// TIA Portal V15.1 export
// export: Created 2020-06-12T07:35:40.5849609Z, ExportSetting None, DisplayName Totally Integrated Automation Portal, DisplayVersion V15.1, DisplayName TIA Portal Openness, DisplayVersion V15.1, DisplayName STEP 7 Professional, DisplayVersion V15.1, DisplayName STEP 7 Safety, DisplayVersion V15.1, DisplayName WinCC Advanced, DisplayVersion V15.1
FUNCTION_BLOCK "F_call"   // FB3, F_FBD
TITLE = Failsafe MAIN program
{ S7_Optimized_Access := 'TRUE' }
   VAR
      emst_del_reset { ExternalAccessible := 'False'; ExternalVisible := 'False'; ExternalWritable := 'False'} : Bool;   // EmStop delayed reset
      ESTOP { ExternalAccessible := 'False'; ExternalVisible := 'False'; ExternalWritable := 'False'} : ESTOP1;
      ACK { ExternalAccessible := 'False'; ExternalVisible := 'False'; ExternalWritable := 'False'} : ACK_GL;
      SD1_TOF { ExternalAccessible := 'False'; ExternalVisible := 'False'; ExternalWritable := 'False'} : TOF;
      RS_TON { ExternalAccessible := 'False'; ExternalVisible := 'False'; ExternalWritable := 'False'} : TON;
      FBACK_EMER_UNDEL { ExternalAccessible := 'False'; ExternalVisible := 'False'; ExternalWritable := 'False'} : FDBACK;
      FBACK_EMER_DEL { ExternalAccessible := 'False'; ExternalVisible := 'False'; ExternalWritable := 'False'} : FDBACK;
      FBACK_ES1LE1_EV02 { ExternalAccessible := 'False'; ExternalVisible := 'False'; ExternalWritable := 'False'} : FDBACK;
      FBACK_ES1LE1_M01 { ExternalAccessible := 'False'; ExternalVisible := 'False'; ExternalWritable := 'False'} : FDBACK;
      FBACK_ES1LE1_M01STO { ExternalAccessible := 'False'; ExternalVisible := 'False'; ExternalWritable := 'False'} : FDBACK;
      FBACK_ES1LE2_M01 { ExternalAccessible := 'False'; ExternalVisible := 'False'; ExternalWritable := 'False'} : FDBACK;
      FBACK_ES1LE2_M02 { ExternalAccessible := 'False'; ExternalVisible := 'False'; ExternalWritable := 'False'} : FDBACK;
      FBACK_ES1LE3_M01 { ExternalAccessible := 'False'; ExternalVisible := 'False'; ExternalWritable := 'False'} : FDBACK;
      FBACK_ES1LE3_M01STO { ExternalAccessible := 'False'; ExternalVisible := 'False'; ExternalWritable := 'False'} : FDBACK;
      FBACK_ES1LE4_EV01 { ExternalAccessible := 'False'; ExternalVisible := 'False'; ExternalWritable := 'False'} : FDBACK;
      FBACK_ES1LE4_EV02 { ExternalAccessible := 'False'; ExternalVisible := 'False'; ExternalWritable := 'False'} : FDBACK;
      FBACK_ES1LE4_M01 { ExternalAccessible := 'False'; ExternalVisible := 'False'; ExternalWritable := 'False'} : FDBACK;
      FBACK_ES1LE4_M01STO { ExternalAccessible := 'False'; ExternalVisible := 'False'; ExternalWritable := 'False'} : FDBACK;
      FBACK_ES1LM1_EV01 { ExternalAccessible := 'False'; ExternalVisible := 'False'; ExternalWritable := 'False'} : FDBACK;
      FBACK_ES1LM2_EV01 { ExternalAccessible := 'False'; ExternalVisible := 'False'; ExternalWritable := 'False'} : FDBACK;
      FBACK_ES1LS1_XS01 { ExternalAccessible := 'False'; ExternalVisible := 'False'; ExternalWritable := 'False'} : FDBACK;
      TOF_GYxx { ExternalAccessible := 'False'; ExternalVisible := 'False'; ExternalWritable := 'False'} : TOF;
      TOF_hood { ExternalAccessible := 'False'; ExternalVisible := 'False'; ExternalWritable := 'False'} : TOF;
      TOF_mcb { ExternalAccessible := 'False'; ExternalVisible := 'False'; ExternalWritable := 'False'} : TOF;
      TOF_trafo { ExternalAccessible := 'False'; ExternalVisible := 'False'; ExternalWritable := 'False'} : TOF;
      TMR_S43_flt { ExternalAccessible := 'False'; ExternalVisible := 'False'; ExternalWritable := 'False'} : TON;
      TMR_S43_auto { ExternalAccessible := 'False'; ExternalVisible := 'False'; ExternalWritable := 'False'} : TOF;
   END_VAR
   VAR_TEMP
      _area_safe : Bool;
      _hood_is_closed : Bool;
      _reset : Bool;
      _del_reset : Bool;
      _GD01_S43_flt : Bool;
      _GD01_S43_off : Bool;
      _GD01_S43_auto : Bool;
   END_VAR
BEGIN

REGION Network 1: Delayed automatic reset by GD01-S34 (timeout)
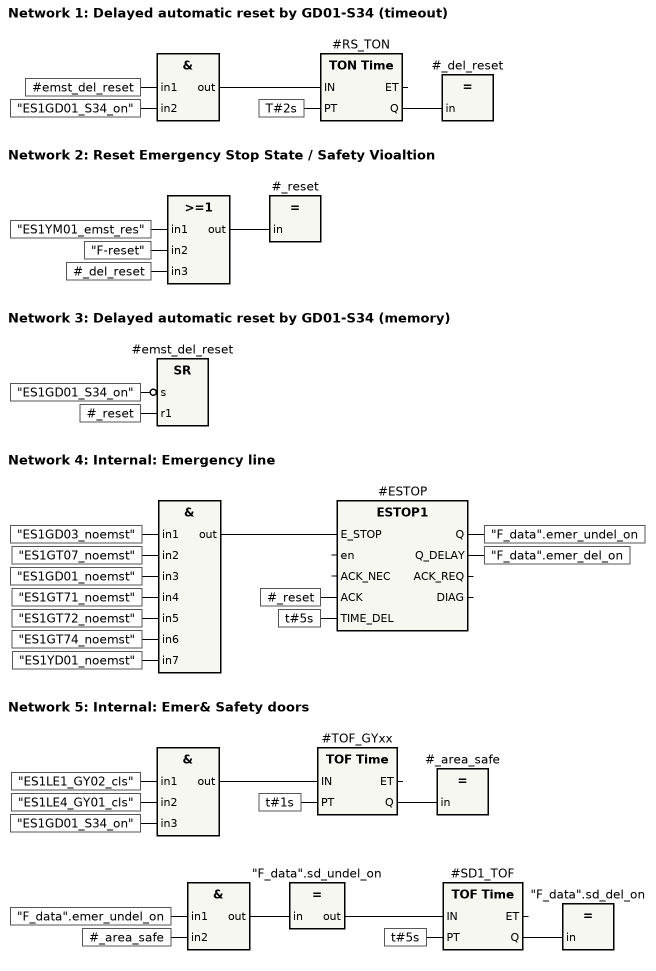
   #RS_TON.TON(IN := #emst_del_reset AND "ES1GD01_S34_on", PT := T#2s);
   #_del_reset := #RS_TON.Q;
END_REGION

REGION Network 2: Reset Emergency Stop State / Safety Vioaltion
   #_reset := "ES1YM01_emst_res" OR "F-reset" OR #_del_reset;
END_REGION

REGION Network 3: Delayed automatic reset by GD01-S34 (memory)
   IF NOT "ES1GD01_S34_on" THEN
       #emst_del_reset := TRUE;   // SR flip-flop
   END_IF;
   IF #_reset THEN #emst_del_reset := FALSE; END_IF;
END_REGION

REGION Network 4: Internal: Emergency line
   #ESTOP(E_STOP := "ES1GD03_noemst" AND "ES1GT07_noemst" AND "ES1GD01_noemst" AND "ES1GT71_noemst" AND "ES1GT72_noemst" AND "ES1GT74_noemst" AND "ES1YD01_noemst",   // ESTOP1
          ACK := #_reset,
          TIME_DEL := t#5s,
          Q => "F_data".emer_undel_on,
          Q_DELAY => "F_data".emer_del_on);
END_REGION

REGION Network 5: Internal: Emer& Safety doors
   // ES1LE1.GY02 = top platfromr safety door
   // ES1LE4.GY01 = portal ladder
   #TOF_GYxx.TOF(IN := "ES1LE1_GY02_cls" AND "ES1LE4_GY01_cls" AND "ES1GD01_S34_on", PT := t#1s);
   #_area_safe := #TOF_GYxx.Q;
   "F_data".sd_undel_on := "F_data".emer_undel_on AND #_area_safe;
   #SD1_TOF.TOF(IN := "F_data".sd_undel_on, PT := t#5s);
   "F_data".sd_del_on := #SD1_TOF.Q;
END_REGION

REGION Network 6: ES1GD01-S43 treat
   // The switch S43 has non-ideal switching: the signal between positions are all 0
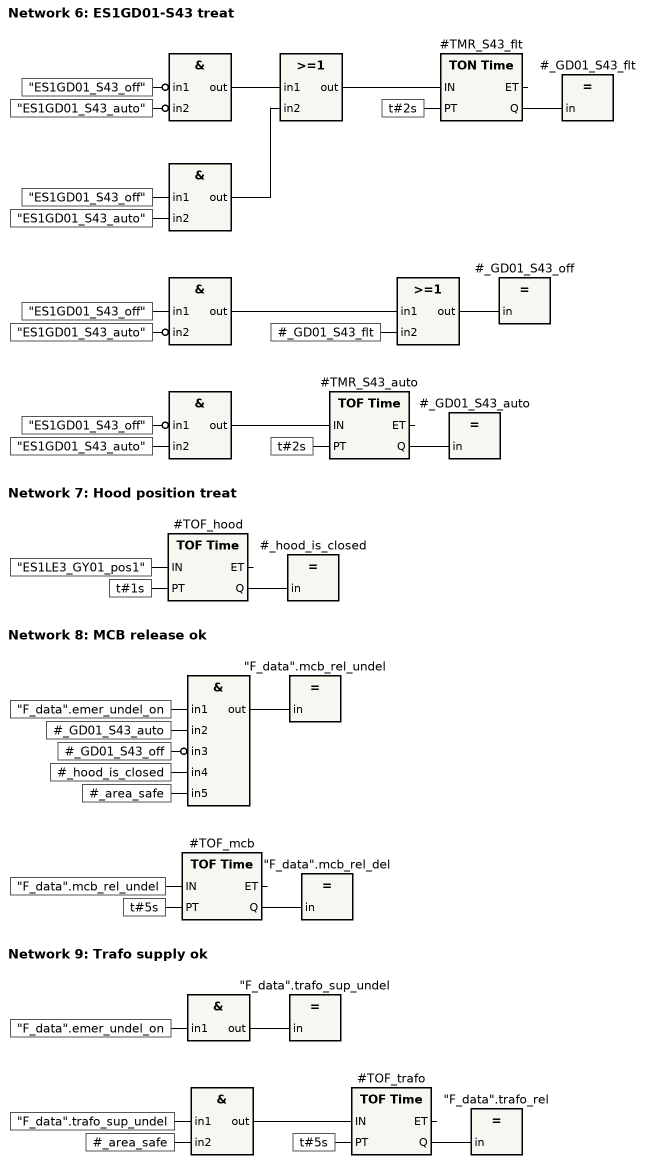
   #TMR_S43_flt.TON(IN := (NOT "ES1GD01_S43_off" AND NOT "ES1GD01_S43_auto") OR ("ES1GD01_S43_off" AND "ES1GD01_S43_auto"),
                    PT := t#2s);
   #_GD01_S43_flt := #TMR_S43_flt.Q;
   #_GD01_S43_off := ("ES1GD01_S43_off" AND NOT "ES1GD01_S43_auto") OR #_GD01_S43_flt;
   #TMR_S43_auto.TOF(IN := NOT "ES1GD01_S43_off" AND "ES1GD01_S43_auto", PT := t#2s);
   #_GD01_S43_auto := #TMR_S43_auto.Q;
END_REGION

REGION Network 7: Hood position treat
   #TOF_hood.TOF(IN := "ES1LE3_GY01_pos1", PT := t#1s);
   #_hood_is_closed := #TOF_hood.Q;
END_REGION

REGION Network 8: MCB release ok
   "F_data".mcb_rel_undel := "F_data".emer_undel_on AND #_GD01_S43_auto AND NOT #_GD01_S43_off AND #_hood_is_closed AND #_area_safe;
   #TOF_mcb.TOF(IN := "F_data".mcb_rel_undel, PT := t#5s);
   "F_data".mcb_rel_del := #TOF_mcb.Q;
END_REGION

REGION Network 9: Trafo supply ok
   "F_data".trafo_sup_undel := "F_data".emer_undel_on;
   #TOF_trafo.TOF(IN := "F_data".trafo_sup_undel AND #_area_safe, PT := t#5s);
   "F_data".trafo_rel := #TOF_trafo.Q;
END_REGION

REGION Network 10: Out: Emergency line Undelayed
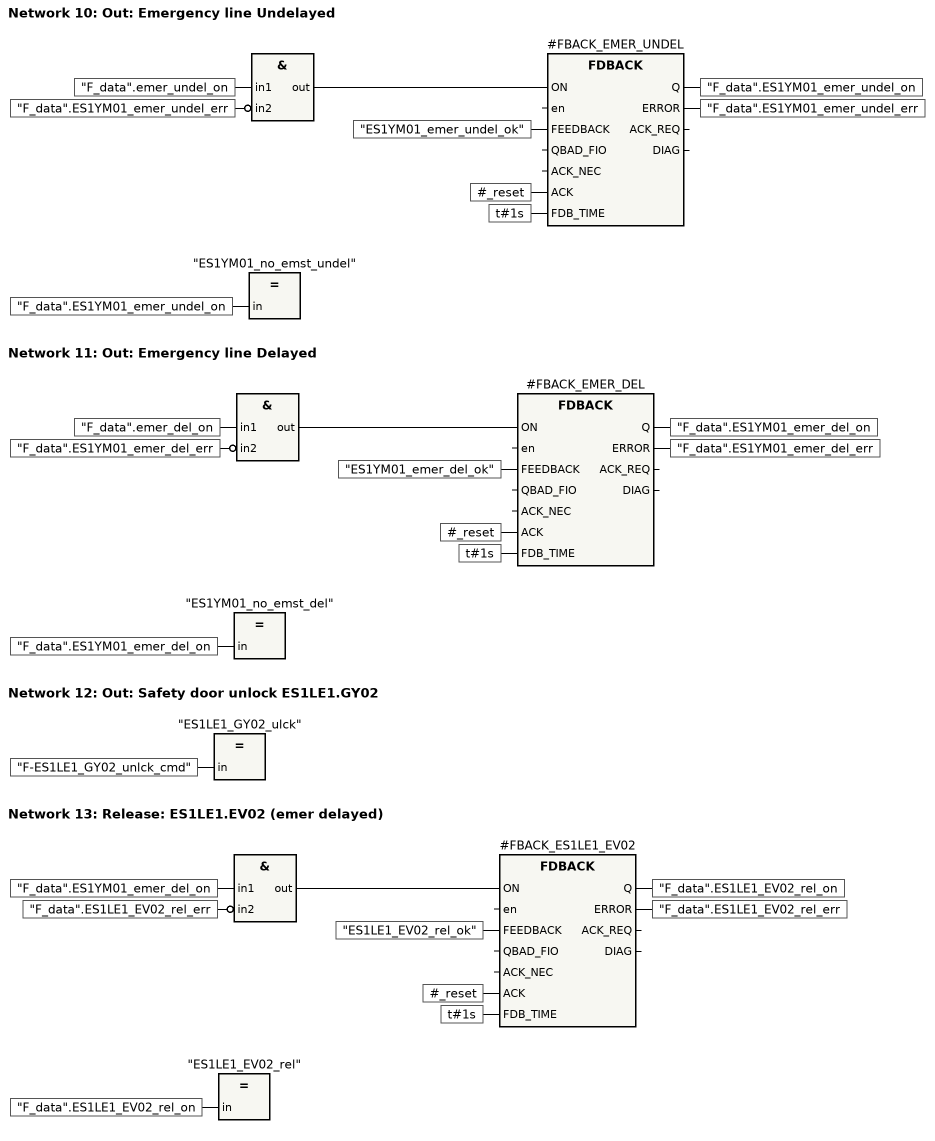
   #FBACK_EMER_UNDEL(ON := "F_data".emer_undel_on AND NOT "F_data".ES1YM01_emer_undel_err,   // FDBACK
                     FEEDBACK := "ES1YM01_emer_undel_ok",
                     ACK := #_reset,
                     FDB_TIME := t#1s,
                     Q => "F_data".ES1YM01_emer_undel_on,
                     ERROR => "F_data".ES1YM01_emer_undel_err);
   "ES1YM01_no_emst_undel" := "F_data".ES1YM01_emer_undel_on;
END_REGION

REGION Network 11: Out: Emergency line Delayed
   #FBACK_EMER_DEL(ON := "F_data".emer_del_on AND NOT "F_data".ES1YM01_emer_del_err,   // FDBACK
                   FEEDBACK := "ES1YM01_emer_del_ok",
                   ACK := #_reset,
                   FDB_TIME := t#1s,
                   Q => "F_data".ES1YM01_emer_del_on,
                   ERROR => "F_data".ES1YM01_emer_del_err);
   "ES1YM01_no_emst_del" := "F_data".ES1YM01_emer_del_on;
END_REGION

REGION Network 12: Out: Safety door unlock ES1LE1.GY02
   "ES1LE1_GY02_ulck" := "F-ES1LE1_GY02_unlck_cmd";
END_REGION

REGION Network 13: Release: ES1LE1.EV02 (emer delayed)
   #FBACK_ES1LE1_EV02(ON := "F_data".ES1YM01_emer_del_on AND NOT "F_data".ES1LE1_EV02_rel_err,   // FDBACK
                      FEEDBACK := "ES1LE1_EV02_rel_ok",
                      ACK := #_reset,
                      FDB_TIME := t#1s,
                      Q => "F_data".ES1LE1_EV02_rel_on,
                      ERROR => "F_data".ES1LE1_EV02_rel_err);
   "ES1LE1_EV02_rel" := "F_data".ES1LE1_EV02_rel_on;
END_REGION

REGION Network 14: Release: ES1LE4.EV01 (emer delayed)
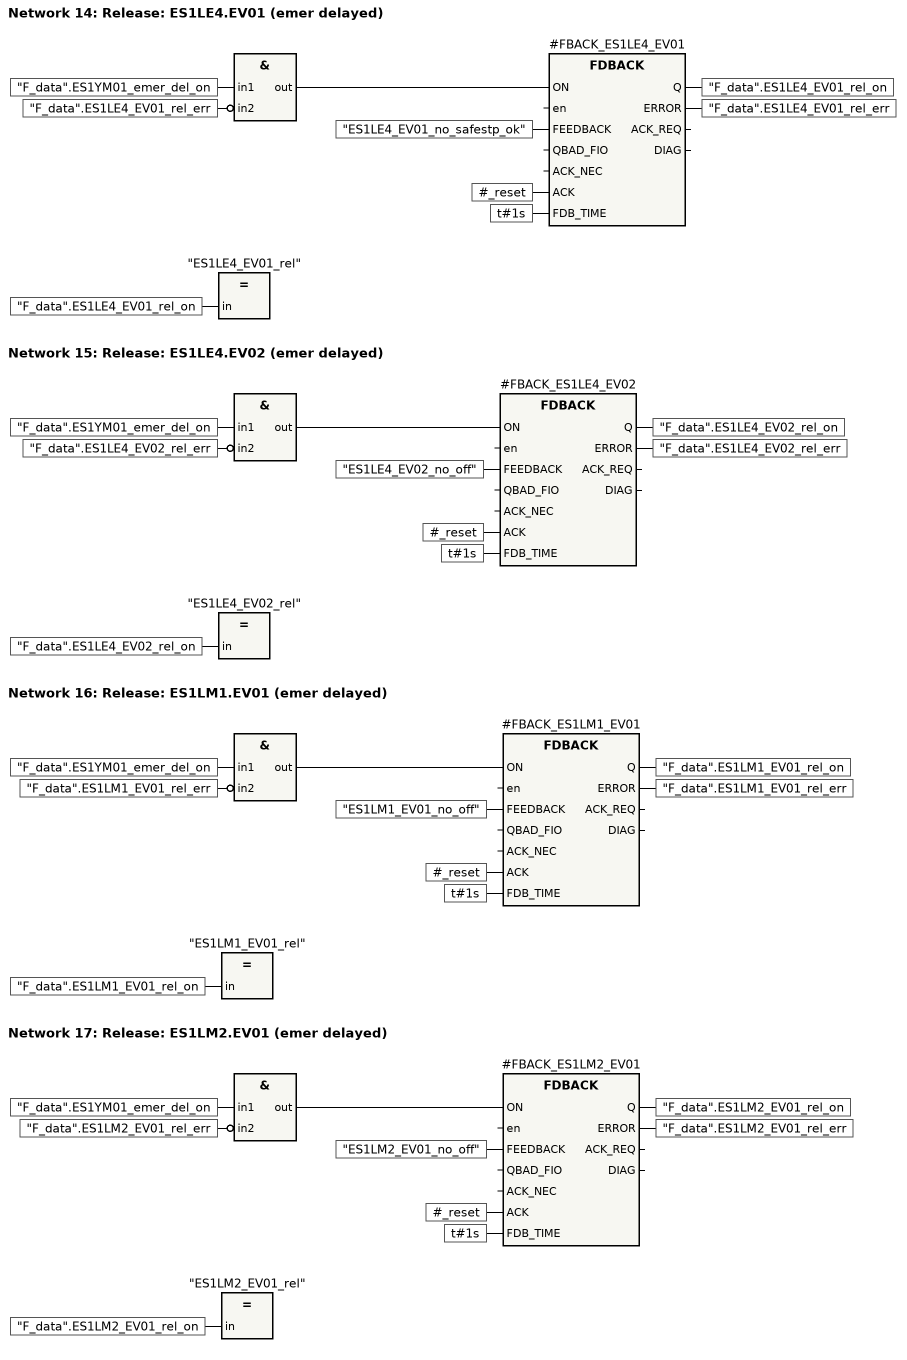
   #FBACK_ES1LE4_EV01(ON := "F_data".ES1YM01_emer_del_on AND NOT "F_data".ES1LE4_EV01_rel_err,   // FDBACK
                      FEEDBACK := "ES1LE4_EV01_no_safestp_ok",
                      ACK := #_reset,
                      FDB_TIME := t#1s,
                      Q => "F_data".ES1LE4_EV01_rel_on,
                      ERROR => "F_data".ES1LE4_EV01_rel_err);
   "ES1LE4_EV01_rel" := "F_data".ES1LE4_EV01_rel_on;
END_REGION

REGION Network 15: Release: ES1LE4.EV02 (emer delayed)
   #FBACK_ES1LE4_EV02(ON := "F_data".ES1YM01_emer_del_on AND NOT "F_data".ES1LE4_EV02_rel_err,   // FDBACK
                      FEEDBACK := "ES1LE4_EV02_no_off",
                      ACK := #_reset,
                      FDB_TIME := t#1s,
                      Q => "F_data".ES1LE4_EV02_rel_on,
                      ERROR => "F_data".ES1LE4_EV02_rel_err);
   "ES1LE4_EV02_rel" := "F_data".ES1LE4_EV02_rel_on;
END_REGION

REGION Network 16: Release: ES1LM1.EV01 (emer delayed)
   #FBACK_ES1LM1_EV01(ON := "F_data".ES1YM01_emer_del_on AND NOT "F_data".ES1LM1_EV01_rel_err,   // FDBACK
                      FEEDBACK := "ES1LM1_EV01_no_off",
                      ACK := #_reset,
                      FDB_TIME := t#1s,
                      Q => "F_data".ES1LM1_EV01_rel_on,
                      ERROR => "F_data".ES1LM1_EV01_rel_err);
   "ES1LM1_EV01_rel" := "F_data".ES1LM1_EV01_rel_on;
END_REGION

REGION Network 17: Release: ES1LM2.EV01 (emer delayed)
   #FBACK_ES1LM2_EV01(ON := "F_data".ES1YM01_emer_del_on AND NOT "F_data".ES1LM2_EV01_rel_err,   // FDBACK
                      FEEDBACK := "ES1LM2_EV01_no_off",
                      ACK := #_reset,
                      FDB_TIME := t#1s,
                      Q => "F_data".ES1LM2_EV01_rel_on,
                      ERROR => "F_data".ES1LM2_EV01_rel_err);
   "ES1LM2_EV01_rel" := "F_data".ES1LM2_EV01_rel_on;
END_REGION

REGION Network 18: Release: ES1LE1.M01 (emer undelayed)
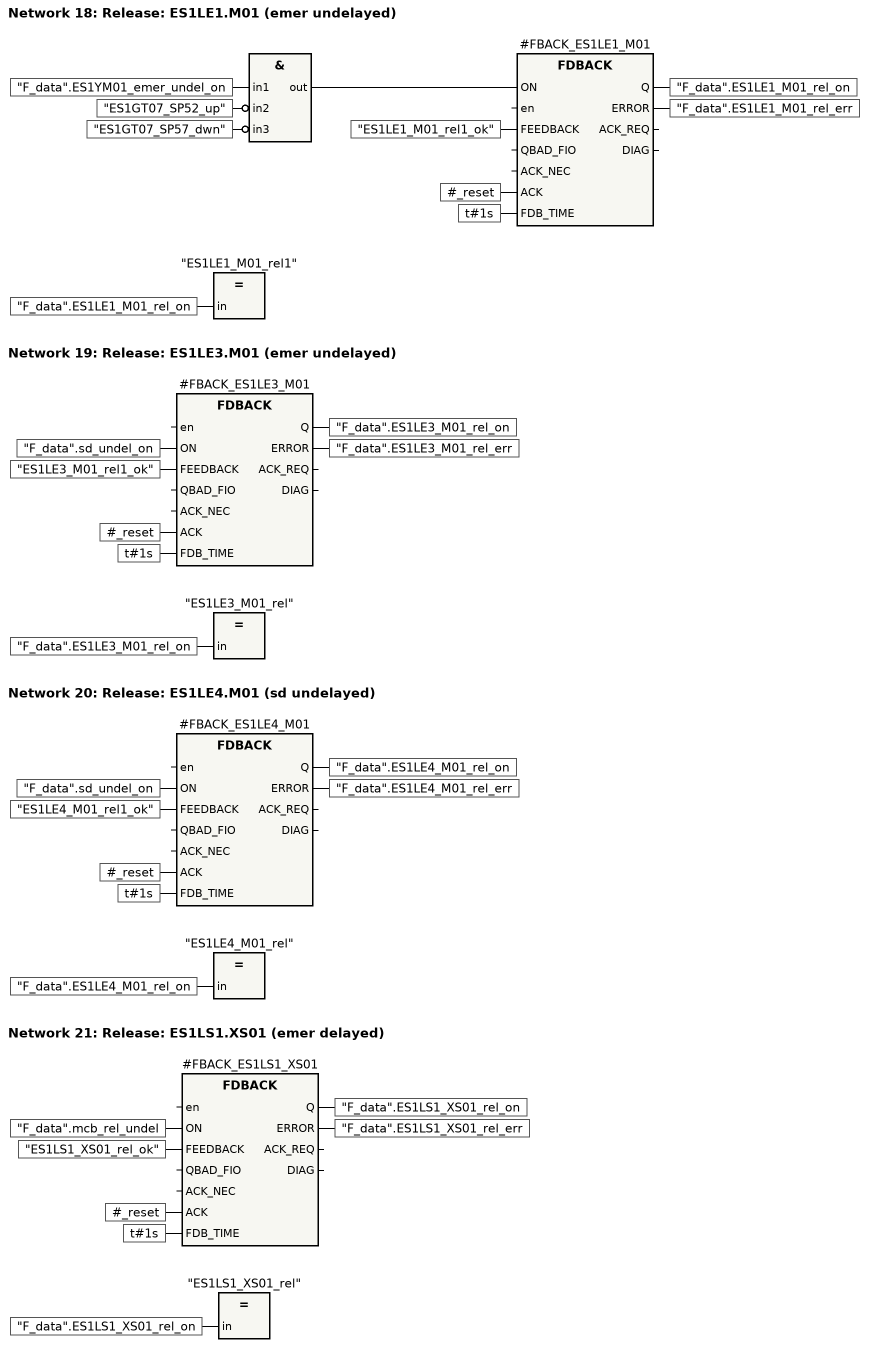
   #FBACK_ES1LE1_M01(ON := "F_data".ES1YM01_emer_undel_on AND NOT "ES1GT07_SP52_up" AND NOT "ES1GT07_SP57_dwn",   // FDBACK
                     FEEDBACK := "ES1LE1_M01_rel1_ok",
                     ACK := #_reset,
                     FDB_TIME := t#1s,
                     Q => "F_data".ES1LE1_M01_rel_on,
                     ERROR => "F_data".ES1LE1_M01_rel_err);
   "ES1LE1_M01_rel1" := "F_data".ES1LE1_M01_rel_on;
END_REGION

REGION Network 19: Release: ES1LE3.M01 (emer undelayed)
   #FBACK_ES1LE3_M01(ON := "F_data".sd_undel_on,   // FDBACK
                     FEEDBACK := "ES1LE3_M01_rel1_ok",
                     ACK := #_reset,
                     FDB_TIME := t#1s,
                     Q => "F_data".ES1LE3_M01_rel_on,
                     ERROR => "F_data".ES1LE3_M01_rel_err);
   "ES1LE3_M01_rel" := "F_data".ES1LE3_M01_rel_on;
END_REGION

REGION Network 20: Release: ES1LE4.M01 (sd undelayed)
   #FBACK_ES1LE4_M01(ON := "F_data".sd_undel_on,   // FDBACK
                     FEEDBACK := "ES1LE4_M01_rel1_ok",
                     ACK := #_reset,
                     FDB_TIME := t#1s,
                     Q => "F_data".ES1LE4_M01_rel_on,
                     ERROR => "F_data".ES1LE4_M01_rel_err);
   "ES1LE4_M01_rel" := "F_data".ES1LE4_M01_rel_on;
END_REGION

REGION Network 21: Release: ES1LS1.XS01 (emer delayed)
   #FBACK_ES1LS1_XS01(ON := "F_data".mcb_rel_undel,   // FDBACK
                      FEEDBACK := "ES1LS1_XS01_rel_ok",
                      ACK := #_reset,
                      FDB_TIME := t#1s,
                      Q => "F_data".ES1LS1_XS01_rel_on,
                      ERROR => "F_data".ES1LS1_XS01_rel_err);
   "ES1LS1_XS01_rel" := "F_data".ES1LS1_XS01_rel_on;
END_REGION

REGION Network 22: Release ES1LT1.XS01/no_emst (emer undelayed)
   // !! WARNING! 
   // PuM/2018-08-13: This E-STOP is not in SafetyMatrix and it has only one line (not two as required). Because of that I implement only local emeregecny stop.
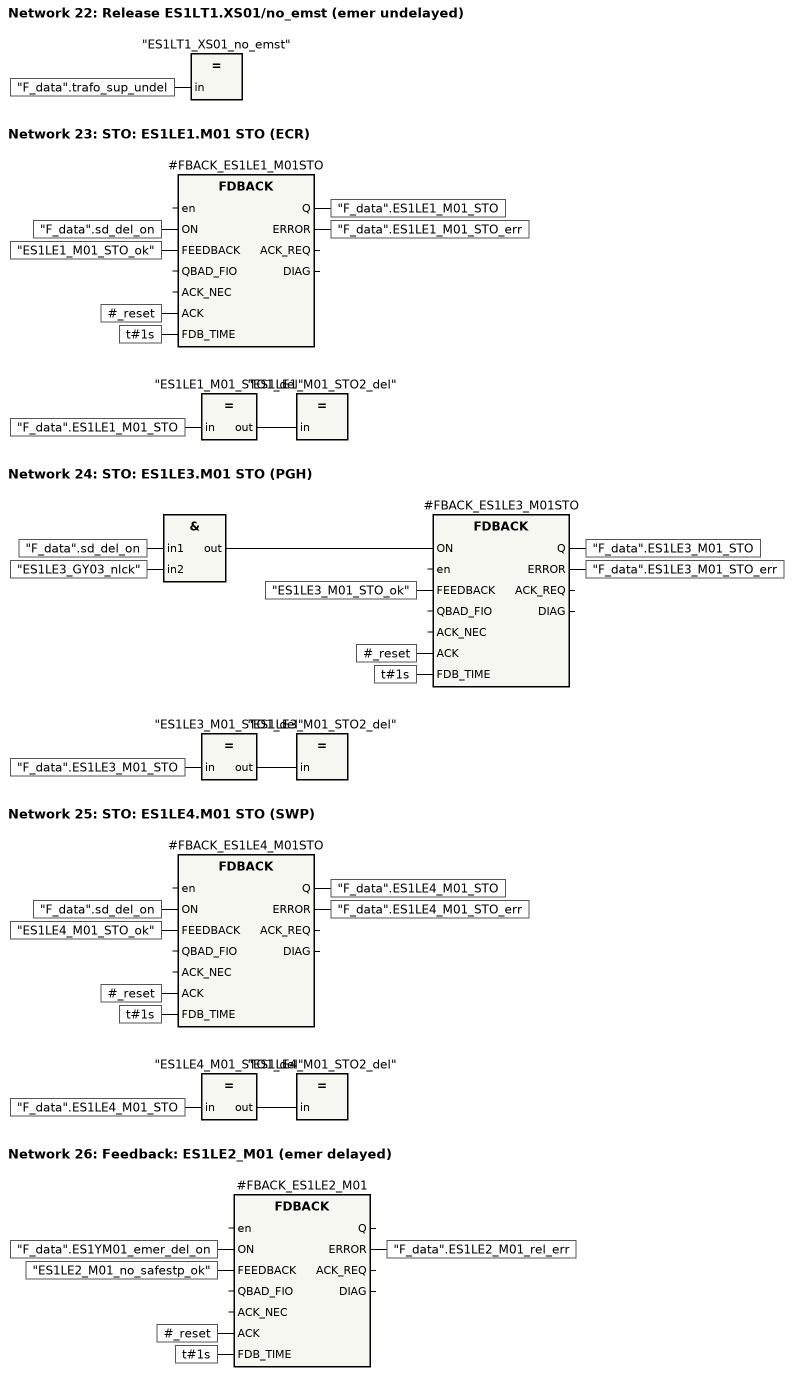
   "ES1LT1_XS01_no_emst" := "F_data".trafo_sup_undel;
END_REGION

REGION Network 23: STO: ES1LE1.M01 STO (ECR)
   #FBACK_ES1LE1_M01STO(ON := "F_data".sd_del_on,   // FDBACK
                        FEEDBACK := "ES1LE1_M01_STO_ok",
                        ACK := #_reset,
                        FDB_TIME := t#1s,
                        Q => "F_data".ES1LE1_M01_STO,
                        ERROR => "F_data".ES1LE1_M01_STO_err);
   "ES1LE1_M01_STO1_del" := "F_data".ES1LE1_M01_STO;
   "ES1LE1_M01_STO2_del" := "F_data".ES1LE1_M01_STO;
END_REGION

REGION Network 24: STO: ES1LE3.M01 STO (PGH)
   #FBACK_ES1LE3_M01STO(ON := "F_data".sd_del_on AND "ES1LE3_GY03_nlck",   // FDBACK
                        FEEDBACK := "ES1LE3_M01_STO_ok",
                        ACK := #_reset,
                        FDB_TIME := t#1s,
                        Q => "F_data".ES1LE3_M01_STO,
                        ERROR => "F_data".ES1LE3_M01_STO_err);
   "ES1LE3_M01_STO1_del" := "F_data".ES1LE3_M01_STO;
   "ES1LE3_M01_STO2_del" := "F_data".ES1LE3_M01_STO;
END_REGION

REGION Network 25: STO: ES1LE4.M01 STO (SWP)
   // "F_data".ES1LE4_M01_rel_on
   #FBACK_ES1LE4_M01STO(ON := "F_data".sd_del_on,   // FDBACK
                        FEEDBACK := "ES1LE4_M01_STO_ok",
                        ACK := #_reset,
                        FDB_TIME := t#1s,
                        Q => "F_data".ES1LE4_M01_STO,
                        ERROR => "F_data".ES1LE4_M01_STO_err);
   "ES1LE4_M01_STO1_del" := "F_data".ES1LE4_M01_STO;
   "ES1LE4_M01_STO2_del" := "F_data".ES1LE4_M01_STO;
END_REGION

REGION Network 26: Feedback: ES1LE2_M01 (emer delayed)
   #FBACK_ES1LE2_M01(ON := "F_data".ES1YM01_emer_del_on,   // FDBACK
                     FEEDBACK := "ES1LE2_M01_no_safestp_ok",
                     ACK := #_reset,
                     FDB_TIME := t#1s,
                     ERROR => "F_data".ES1LE2_M01_rel_err);
END_REGION

REGION Network 27: Feedback: ES1LE2_M02 (emer delayed)
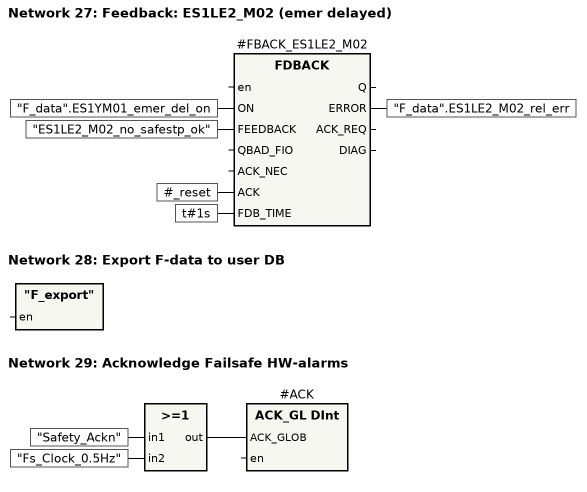
   #FBACK_ES1LE2_M02(ON := "F_data".ES1YM01_emer_del_on,   // FDBACK
                     FEEDBACK := "ES1LE2_M02_no_safestp_ok",
                     ACK := #_reset,
                     FDB_TIME := t#1s,
                     ERROR => "F_data".ES1LE2_M02_rel_err);
END_REGION

REGION Network 28: Export F-data to user DB
   "F_export"();
END_REGION

REGION Network 29: Acknowledge Failsafe HW-alarms
   #ACK(ACK_GLOB := "Safety_Ackn" OR "Fs_Clock_0.5Hz");   // ACK_GL
END_REGION
END_FUNCTION_BLOCK
